FUNCTION_BLOCK NumberEdit
VAR
	_number : REAL;
END_VAR

PROPERTY Number : REAL
GET
Number := _number;
END_GET
SET
_number := Number;
END_SET
END_PROPERTY

END_FUNCTION_BLOCK

(* stored: Version 1.1.0.1, ProductVersion 3.1.4024.12
   POU NumberEdit: Id {dd182afd-7d10-410a-9d00-31674a3839a1}, SpecialFunc None
   Property Number: Id {8682b28b-7865-4c12-826a-43e63df61efb}
   Get Get: Id {7bf59276-0c37-4650-94d1-3c8840a47970}
   Set Set: Id {402c2567-9276-4a34-9b14-1d907f6e18f8} *)
